{attribute 'qualified_only'}
{attribute 'strict'}
TYPE eGenControlProtocol :
(
	None := 0,
	AGC150 := 1
);
END_TYPE

(* stored: Version 1.1.0.1, ProductVersion 3.1.4026.18
   DUT eGenControlProtocol: Id {1e05eceb-9c90-46bb-932c-30c7d6153eed} *)
